(* IEC 61131-3 sources: ieccompiler/test/syn_tests/exceptions, 9 files *)

(* ---- test_fun_argsassignment.st ---- *)
FUNCTION test_fun_argsassignment:INT
  VAR
    KK:INT;
    VV:BOOL;
  END_VAR

  VAR_INPUT
    BBB:INT;
    CCC:INT;
  END_VAR

  CCC := BBB + CCC + 9;
END_FUNCTION

(* ---- test_fb_call.st ---- *)
PROGRAM test_fb_call
  VAR
    fb : TestFb;
  END_VAR
  fb(TRUE, 12, 13);

END_PROGRAM

FUNCTION_BLOCK test_fb_define
  VAR_INPUT
    bFlag:BOOL;
    A:INT;
    B:INT;
  END_VAR
END_FUNCTION_BLOCK

(* ---- test_fun_args.st ---- *)
PROGRAM test_fun_args
  VAR
    B:INT;
    C:INT;
    D:BOOL;
  END_VAR

  C:=test_fun_args_add(B);
END_PROGRAM

FUNCTION test_fun_args_add:INT
  VAR
    KK:INT;
    VV:BOOL;
  END_VAR

  VAR_INPUT
    BBB:INT;
    CCC:INT;
  END_VAR

  KK := BBB + CCC + 9;
END_FUNCTION

(* ---- test_if_abn.st ---- *)
PROGRAM test_if_abn
  VAR
    b_Start_Stop:DINT;
    N:DINT;
  END_VAR

  IF b_Start_Stop > 0 THEN
    N := N + 7;
  END_IF
END_PROGRAM

(* ---- test_repeat_abn1.st ---- *)
PROGRAM test_repeat_abn1
  VAR
    i  : INT;
  END_VAR

  REPEAT
    i := i + 1;
  UNTIL i = 4;
  END_REPEAT
END_PROGRAM

(* ---- test_while_abn1.st ---- *)
PROGRAM test_while_abn1
  VAR
    b_Start_Stop:DINT;
    N:DINT;
  END_VAR

  WHILE b_Start_Stop > 111111 OR N < 222222
    N := N + 7;
  END_WHILE
END_PROGRAM

(* ---- test_while_abn2.st ---- *)
PROGRAM test_while_abn2
  VAR
    b_Start_Stop:DINT;
    N:DINT;
  END_VAR

  WHILE b_Start_Stop > 111111 OR N < 222222 DO
    N := N + 7
  END_WHILE
END_PROGRAM

(* ---- test_while_abn3.st ---- *)
PROGRAM test_while_abn3
  VAR
    b_Start_Stop:DINT;
    N:DINT;
  END_VAR

  WHILE b_Start_Stop > 111111 OR N < 222222 DO
    N := N + 7;
  END_WHILE;
END_PROGRAM

(* ---- test_while_abn4.st ---- *)
PROGRAM test_while_abn4
  VAR
    b_Start_Stop:DINT;
    N:DINT;
  END_VAR

  WHILE b_Start_Stop > 111111 OR N < 222222 DO
    N := N + 7;
  END_WHILE

  WHILE b_Start_Stop > 111111 AND N < 222222 DO
    N := N + 8;
  END_WHILE

  WHILE b_Start_Stop < 100 OR (b_Start_Stop > 111111 AND b_Start_Stop < 222222)  DO
    N := N + 9;
  END_WHILE

  WHILE b_Start_Stop  > 200 AND (b_Start_Stop < 111111 OR N < 222222 ) DO
    N := N + 10;
  END_WHILE
END_PROGRAM
